{attribute 'linkalways'} 
{attribute 'no_explicit_call' := 'This FB is a CLASS and must be accessed using methods or properties'}
{attribute 'enable_dynamic_creation'}
FUNCTION_BLOCK MockAliasDatatype_HRESULT EXTENDS AliasDatatypeBase
VAR
	localData : HRESULT;
	activeData : REFERENCE TO HRESULT REF= localData;
	aliasBaseDatatype : _DINT(localData);
END_VAR

PROPERTY PUBLIC Address : PVOID
GET
Address := ADR(activeData);
END_GET
END_PROPERTY

METHOD PUBLIC ClearReference
VAR_INPUT
END_VAR
activeData REF= localData;
SetBaseDatatypeReference();
END_METHOD

METHOD PUBLIC Clone : I_Datatype
VAR
    pClone : POINTER TO MockAliasDatatype_HRESULT;
END_VAR
pClone := __NEW(MockAliasDatatype_HRESULT(InitialValue := Value));
Clone := pClone^;
END_METHOD

METHOD FB_init : BOOL
VAR_INPUT
	bInitRetains : BOOL; // if TRUE, the retain variables are initialized (warm start / cold start)
	bInCopyCode : BOOL;  // if TRUE, the instance afterwards gets moved into the copy code (online change)
	InitialValue : HRESULT;
END_VAR
localData := InitialValue;
SetBaseDatatypeReference();
AddBaseDatatype(aliasBaseDatatype);
END_METHOD

PROPERTY PUBLIC Identifier : T_MAXSTRING
GET
Identifier := 'HRESULT';
END_GET
END_PROPERTY

METHOD PUBLIC MakeReferenceTo
VAR_INPUT
	ReferenceTarget : REFERENCE TO HRESULT;
END_VAR
activeData REF= ReferenceTarget;
SetBaseDatatypeReference();
END_METHOD

METHOD PROTECTED SetBaseDatatypeReference
VAR_INPUT
END_VAR
aliasBaseDatatype.MakeReferenceTo(activeData);
END_METHOD

PROPERTY PUBLIC Size : UDINT
GET
Size := SIZEOF(activeData);
END_GET
END_PROPERTY

METHOD TryMakeReferenceTo : BOOL
VAR_INPUT
	Target : I_Datatype;
END_VAR
VAR
	targetAsAlias : I_AliasDatatype;
	pTargetData : POINTER TO HRESULT;
END_VAR
IF NOT Target.TryResolveAsAliasDatatype(targetAsAlias) THEN
	RETURN;
END_IF

IF targetAsAlias.Identifier <> Identifier THEN
	RETURN;
END_IF

pTargetData := Target.Address;
activeData REF= pTargetData^;
SetBaseDatatypeReference();
TryMakeReferenceTo := TRUE;
END_METHOD

PROPERTY PUBLIC Value : REFERENCE TO HRESULT
GET
Value REF= activeData;
END_GET
END_PROPERTY

END_FUNCTION_BLOCK

(* stored: Version 1.1.0.1, ProductVersion 3.1.4024.12
   POU MockAliasDatatype_HRESULT: Id {c45195f3-04a5-472c-8341-43ec4284fdcd}, SpecialFunc None
   Folder Constructor: Id {68b0cd46-afa2-4b59-a58b-fe0ffde00f0d}
   Folder Protected: Id {968dd6b6-766c-46be-8c65-33ebe86bb9ea}
   Property Address: Id {6946e33c-787c-4520-926e-cf260ce116ee}
   Get Get: Id {3563c2cc-4851-406d-a2cf-00e0f1a5bcfb}
   Method ClearReference: Id {89dde7fc-d9b3-4b13-ab25-506fd7214d6f}
   Method Clone: Id {3bc5ccc6-d123-4a12-b11e-fba37035742d}
   Method FB_init: Id {2f01bf2d-8043-4f71-b2af-a2de2b91c1e2}
   Property Identifier: Id {773ac119-93ee-466c-b539-188194534577}
   Get Get: Id {a7104f8a-a32b-4f02-af14-2a527152f6c1}
   Method MakeReferenceTo: Id {3f8b1791-7e00-4a92-a33e-bfd815ec9485}
   Method SetBaseDatatypeReference: Id {21ca45a7-7ceb-4b14-a248-587e12870c38}
   Property Size: Id {198cd5cc-fd75-4ee0-8b21-07cba2f48c65}
   Get Get: Id {d51648bc-6c7b-4f21-b5a7-4b4c3f4cb099}
   Method TryMakeReferenceTo: Id {f8c03ec2-690a-4bf4-b597-810db83c41d9}
   Property Value: Id {d059b278-740d-4b19-96d2-454596810b54}
   Get Get: Id {15dfd465-7025-4597-9083-759c58b313da} *)
